// Mitsubishi GX Works2 project: hung_creat_plc_dich_bit_ver2   PLC: FX3U/FX3UC

PROGRAM MAIN
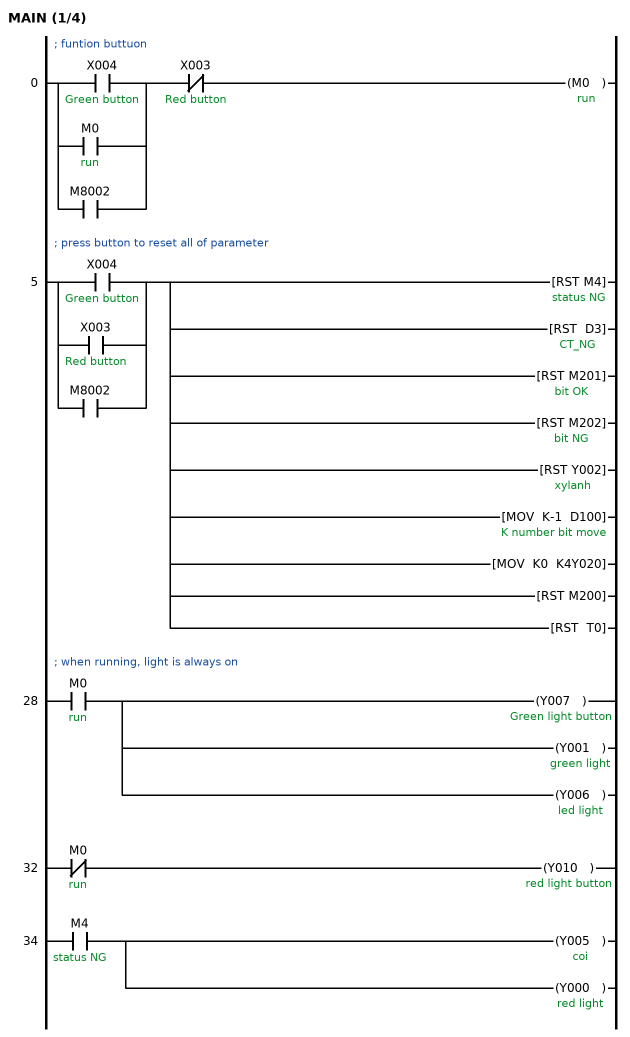
; funtion buttuon
0     LD      X004  ; Green button
      OR      M0  ; run
      OR      M8002
      ANI     X003  ; Red button
      OUT     M0  ; run
; press button to reset all of parameter
5     LD      X004  ; Green button
      OR      X003  ; Red button
      OR      M8002
      RST     M4  ; status NG
      RST     D3  ; CT_NG
      RST     M201  ; bit OK
      RST     M202  ; bit NG
      RST     Y002  ; xylanh
      MOV     K-1 D100  ; K number bit move
      MOV     K0 K4Y020  ; move right
      RST     M200
      RST     T0
; when running, light is always on
28    LD      M0  ; run
      OUT     Y007  ; Green light button
      OUT     Y001  ; green light
      OUT     Y006  ; led light
32    LDI     M0  ; run
      OUT     Y010  ; red light button
34    LD      M4  ; status NG
      OUT     Y005  ; coi
      OUT     Y000  ; red light
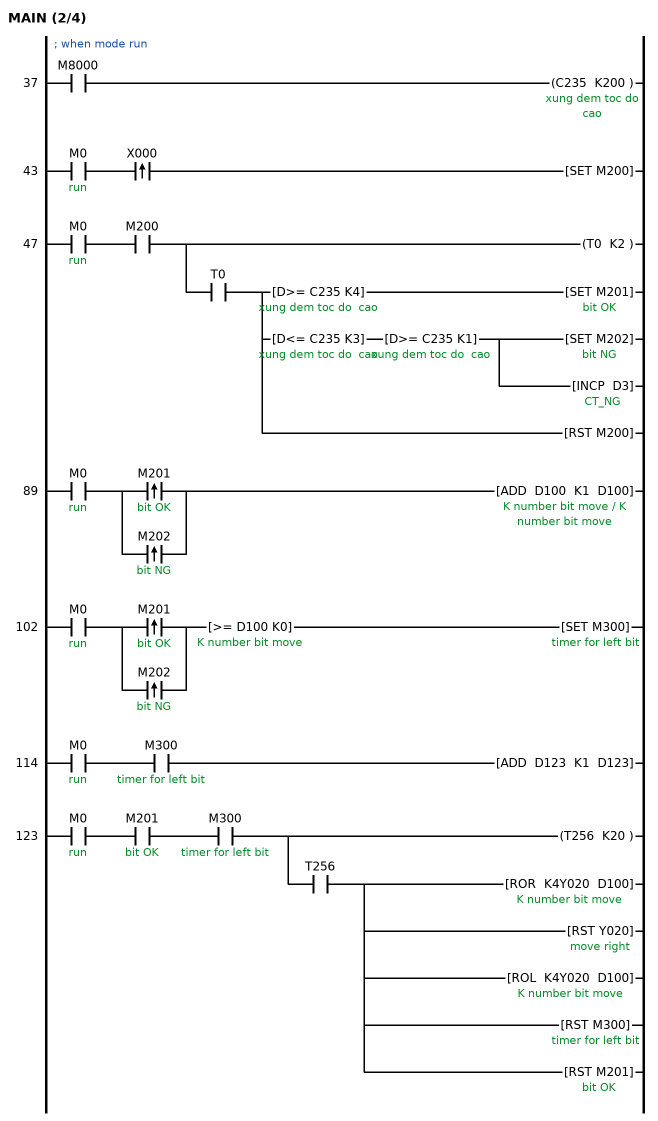
; when mode run
37    LD      M8000
      OUT     C235 K200  ; xung dem toc do  cao
43    LD      M0  ; run
      ANDP    X000
      SET     M200
47    LD      M0  ; run
      AND     M200
      OUT     T0 K2
      AND     T0
      MPS
      ANDD>=  C235 K4  ; xung dem toc do  cao
      SET     M201  ; bit OK
      MRD
      ANDD<=  C235 K3  ; xung dem toc do  cao
      ANDD>=  C235 K1  ; xung dem toc do  cao
      SET     M202  ; bit NG
      INCP    D3
      MPP
      RST     M200
89    LD      M0  ; run
      LDP     M201  ; bit OK
      ORP     M202  ; bit NG
      ANB
      ADD     D100 K1 D100
102   LD      M0  ; run
      LDP     M201  ; bit OK
      ORP     M202  ; bit NG
      ANB
      AND>=   D100 K0  ; K number bit move
      SET     M300  ; timer for left bit
114   LD      M0  ; run
      AND     M300  ; timer for left bit
      ADD     D123 K1 D123
123   LD      M0  ; run
      AND     M201  ; bit OK
      AND     M300  ; timer for left bit
      OUT     T256 K20
      AND     T256
      ROR     K4Y020 D100
      RST     Y020  ; move right
      ROL     K4Y020 D100
      RST     M300  ; timer for left bit
      RST     M201  ; bit OK
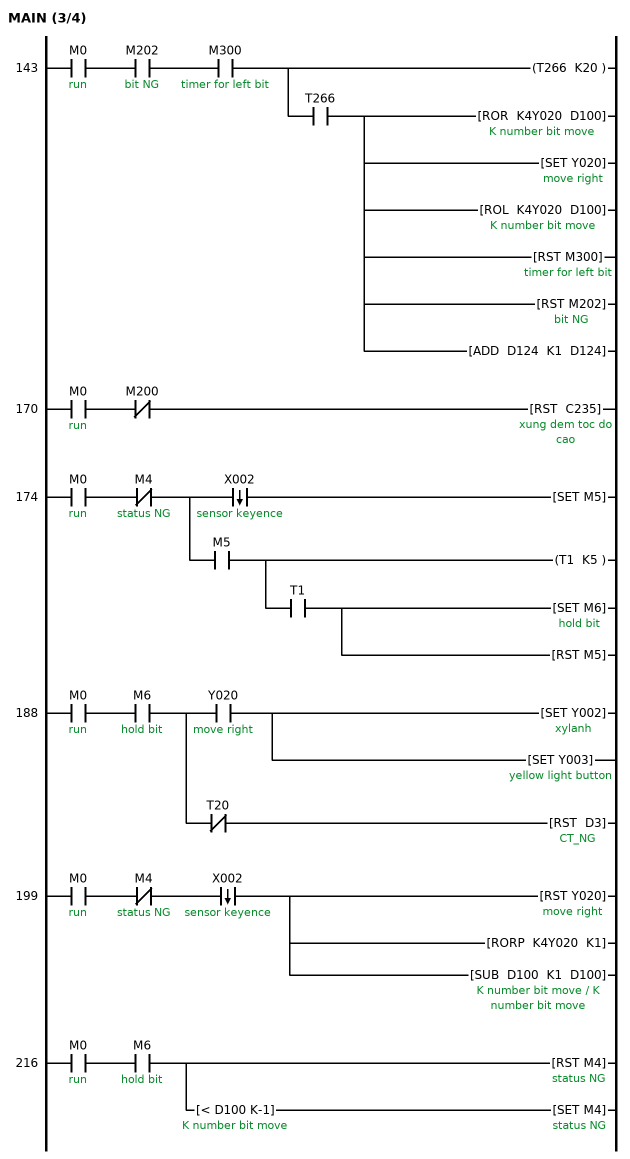
143   LD      M0  ; run
      AND     M202  ; bit NG
      AND     M300  ; timer for left bit
      OUT     T266 K20
      AND     T266
      ROR     K4Y020 D100
      SET     Y020  ; move right
      ROL     K4Y020 D100
      RST     M300  ; timer for left bit
      RST     M202  ; bit NG
      ADD     D124 K1 D124
170   LD      M0  ; run
      ANI     M200
      RST     C235  ; xung dem toc do  cao
174   LD      M0  ; run
      ANI     M4  ; status NG
      MPS
      ANDF    X002  ; sensor keyence
      SET     M5
      MPP
      AND     M5
      OUT     T1 K5
      AND     T1
      SET     M6  ; hold bit
      RST     M5
188   LD      M0  ; run
      AND     M6  ; hold bit
      MPS
      AND     Y020  ; move right
      SET     Y002  ; xylanh
      SET     Y003  ; yellow light button
      MPP
      ANI     T20
      RST     D3  ; CT_NG
199   LD      M0  ; run
      ANI     M4  ; status NG
      ANDF    X002  ; sensor keyence
      RST     Y020  ; move right
      RORP    K4Y020 K1
      SUB     D100 K1 D100
216   LD      M0  ; run
      AND     M6  ; hold bit
      RST     M4  ; status NG
      AND<    D100 K-1  ; K number bit move
      SET     M4  ; status NG
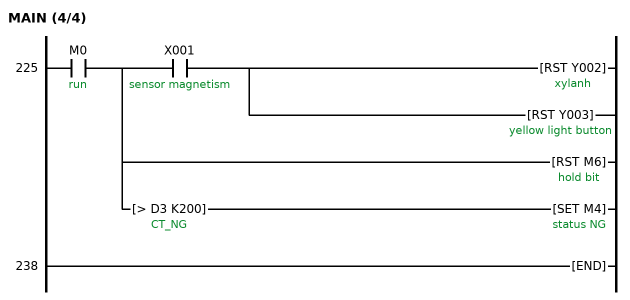
225   LD      M0  ; run
      MPS
      AND     X001  ; sensor magnetism
      RST     Y002  ; xylanh
      RST     Y003  ; yellow light button
      MPP
      RST     M6  ; hold bit
      AND>    D3 K200  ; CT_NG
      SET     M4  ; status NG
238   END
END_PROGRAM

// device comments not shown above
D0  ; CT
M3  ; bit reset NG and OK
M100  ; BIT TO MOVE
